// TIA Portal V20 export
DATA_BLOCK "SBK06"   // DB210
// stored: MemoryReserve 100
   VAR
      "X1-0 Gate EC.Top Close" : Bool;
      "X2-1 Gate EC.LH Close" : Bool;
      "X3-2 Gate EC.RH Close" : Bool;
      "X4-3 reserved" : Bool;
      "X1-4 Gate EC.Top Close" : Bool;
      "X2-5 Gate EC.LH Close" : Bool;
      "X3-6 Gate EC.RH Close" : Bool;
      "X4-7 reserved" : Bool;
      "X5-0 Gate EC.Top UnLock" : Bool;
      "X6-1 Gate EC.LH UnLock" : Bool;
      "X7-2 Gate EC.RH UnLock" : Bool;
   END_VAR
BEGIN
END_DATA_BLOCK
